# EPICS substitutions: evrSupport/Db/ioc/IOC-IN20-AM01trig.substitutions
# Trigger records
#
# refer to Sharepoint document: Controls | Timing | timingTriggers.xls
#
# Must also have pattern records
# Note: WID, DES, TEC are in terms of nSec and are unique per device
#
file evrDevTrig.db {
#      Device	      , Description   , EVR  ,  width ,desired  , EC delay   , EVR  , EVR,  IOC          , slope
#			                            Trigger       wrt TREF   wrt fiducial loca   unit                 1/119Mhz
  pattern { DEV       ,  DESC         , T    ,  WID   , DES     , TEC        , LOCA , UNIT, IOC          , ESLO
                      ,  PREC         , EGU  ,  DRVL  , DRVH    }
	  { LENS:IN20:265:,  "CRG1"       , 0    ,  100   , 10      , 0.1E06     , IN20 , AM01, IOC:IN20:AM01, 8.40336692324359
                      ,  1            ,"nSec", -2.8E06, 2.8E06  }
	  { LENS:IN20:280:,  "CR01"       , 1    ,  100   , 10      , 0.1E06     , IN20 , AM01, IOC:IN20:AM01, 8.40336692324359
                      ,  1            ,"nSec", -2.8E06, 2.8E06  }
}
